{attribute 'GeneratedUsingTerminal: EK1122-0000-0018'}
{attribute addProperty BoxType "EK1122-0000-0018"}
{attribute addProperty Id "Beckhoff_EL9xxxsub_EK1100EK1100_AB5A94672"}
{attribute addProperty CRC "3809521173"}
{attribute addProperty Size "2"}
TYPE Beckhoff_EL9xxxEK1122_E310AE15 EXTENDS EK1122_AB5A9467 :
STRUCT
	{attribute addProperty Name "Beckhoff_EL9xxxsub_EK1100"}
	Beckhoff_EL9xxxsub_EK1100 : EK1100_AB5A9467;
END_STRUCT
END_TYPE

(* stored: Version 1.2.0.0, ProductVersion 3.1.4024.9
   DUT Beckhoff_EL9xxxEK1122_E310AE15: Id {b66a84db-3b48-4e3f-83c6-afa6be76a2f7} *)
